// TIA Portal V17 export
// export: Created 2023-05-07T12:12:08.52961Z, ExportSetting WithDefaults, DisplayName Totally Integrated Automation Portal, DisplayVersion V17, DisplayName TIA Portal Openness, DisplayVersion V17, DisplayName TIA Portal Version Control Interface, DisplayVersion V17, DisplayName TIA Portal Test Suite Advanced, DisplayVersion V17, DisplayName STEP 7 Professional, DisplayVersion V17, DisplayName SIMATIC Energy Suite, DisplayVersion V17, DisplayName STEP 7 Safety, DisplayVersion V17, DisplayName WinCC Professional, DisplayVersion V17
FUNCTION_BLOCK "RAMP"   // FB8, LAD
TITLE = RAMP
{ S7_Optimized_Access := 'TRUE' }
VERSION : 0.1
// stored: AutoNumber true, IsIECCheckEnabled false, IsRetainMemResEnabled false, MemoryReserve 100, SetENOAutomatically false, UDAEnableTagReadback false
   VAR_INPUT
      SetPoint : Real;
      Rate : Real;
      Reset : Bool;
   END_VAR
   VAR_OUTPUT
      OUT : Real := 0.0;
   END_VAR
   VAR
      TON_1 { ExternalAccessible := 'False'; ExternalVisible := 'False'; ExternalWritable := 'False'} : TON_TIME;
      RateDIV : Real;
      Q : Bool;
   END_VAR
   VAR_TEMP   // added for the SCL form of the ladder/FBD networks
      _w1 : Bool;
   END_VAR
BEGIN

REGION Network 1: DIV: Rate/10
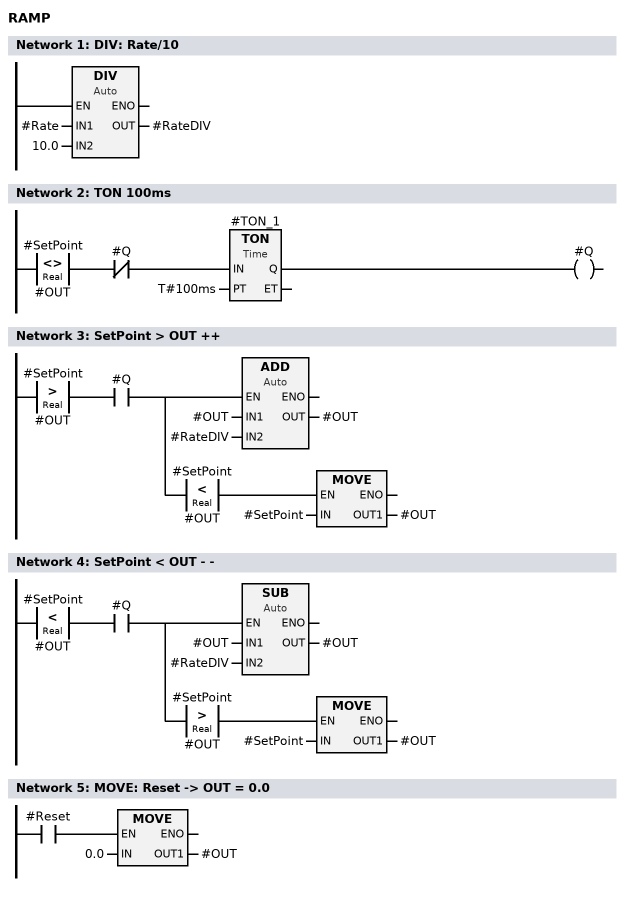
   RUNG wire#powerrail
      Div(in1 := #Rate, in2 := 10.0, out => #RateDIV)
   END_RUNG
   // the same network as SCL:
   #RateDIV := #Rate / 10.0;
END_REGION

REGION Network 2: TON 100ms
   RUNG wire#powerrail
      { S7_Templates := "SrcType := Real" } NE_Contact(in1 := #SetPoint, in2 := #OUT)
      I_Contact( #Q )
      { S7_Templates := "time_type := Time" } #TON_1.TON(pt := T#100ms, et =>)
      Coil( #Q )
   END_RUNG
   // the same network as SCL:
   #TON_1(IN := (#SetPoint <> #OUT) AND NOT #Q, PT := T#100ms);   // TON
   #Q := #TON_1.Q;
END_REGION

REGION Network 3: SetPoint > OUT ++
   RUNG wire#powerrail
      { S7_Templates := "SrcType := Real" } GT_Contact(in1 := #SetPoint, in2 := #OUT)
      Contact( #Q )
      wire#w1
      Add(in1 := #OUT, in2 := #RateDIV, out => #OUT)
   END_RUNG
   RUNG wire#w1
      { S7_Templates := "SrcType := Real" } LT_Contact(in1 := #SetPoint, in2 := #OUT)
      Move(in := #SetPoint, out1 => #OUT)
   END_RUNG
   // the same network as SCL:
   #_w1 := (#SetPoint > #OUT) AND #Q;
   IF #_w1 THEN #OUT := #OUT + #RateDIV; END_IF;
   IF #_w1 AND (#SetPoint < #OUT) THEN #OUT := #SetPoint; END_IF;
END_REGION

REGION Network 4: SetPoint < OUT - -
   RUNG wire#powerrail
      { S7_Templates := "SrcType := Real" } LT_Contact(in1 := #SetPoint, in2 := #OUT)
      Contact( #Q )
      wire#w1
      Sub(in1 := #OUT, in2 := #RateDIV, out => #OUT)
   END_RUNG
   RUNG wire#w1
      { S7_Templates := "SrcType := Real" } GT_Contact(in1 := #SetPoint, in2 := #OUT)
      Move(in := #SetPoint, out1 => #OUT)
   END_RUNG
   // the same network as SCL:
   #_w1 := (#SetPoint < #OUT) AND #Q;
   IF #_w1 THEN #OUT := #OUT - #RateDIV; END_IF;
   IF #_w1 AND (#SetPoint > #OUT) THEN #OUT := #SetPoint; END_IF;
END_REGION

REGION Network 5: MOVE: Reset -> OUT = 0.0
   RUNG wire#powerrail
      Contact( #Reset )
      Move(in := 0.0, out1 => #OUT)
   END_RUNG
   // the same network as SCL:
   IF #Reset THEN #OUT := 0.0; END_IF;
END_REGION
END_FUNCTION_BLOCK
